FUNCTION TFCodicePaccoPresenteInFormaturaAll : BOOL // Se TRUE: codice del pacco presente in formatura, Se FALSE: codice non presente in formatura
VAR_INPUT
	Forming : POINTER TO ARRAY [1..MAXFORMING] OF TFMachinePalletizer_Forming; // Struttura formatura
	CodiceInValutazione : INT; //Codice del pacco da valutare
END_VAR
VAR
	IndiceFormatura : INT;		// Indice della formatura da valutare
	pp : INT;
END_VAR
// Se TRUE: codice del pacco presente in formatura, FALSE: codice non presente in formatura

// Se TRUE: codice del pacco presente in formatura, Se FALSE: codice non presente in formatura
TFCodicePaccoPresenteInFormaturaAll := FALSE;
FOR IndiceFormatura:=1 TO MAXFORMING DO
	IF Forming^[IndiceFormatura].Enable = 1 THEN
		(* Per tutti i codici di Pallettizzazione Validi *)		
		FOR pp:=1 TO MAXFORMINGCODE DO
			IF Forming^[IndiceFormatura].Code[pp] = CodiceInValutazione THEN
				TFCodicePaccoPresenteInFormaturaAll := TRUE;
				RETURN;
			END_IF
		END_FOR
	END_IF
END_FOR

END_FUNCTION

(* stored: Version 1.1.0.1, ProductVersion 3.1.4024.11
   POU TFCodicePaccoPresenteInFormaturaAll: Id {4030ea4e-e652-44da-a0b2-72660ff1563d}, SpecialFunc None *)
